// TIA Portal V17 export
// export: Created 2025-08-05T09:36:00.5262225Z, ExportSetting WithDefaults, DisplayName Totally Integrated Automation Portal, DisplayVersion V17, DisplayName TIA Portal Openness, DisplayVersion V17, DisplayName TIA Portal Version Control Interface, DisplayVersion V17, DisplayName SINAMICS Startdrive Advanced, DisplayVersion V17, DisplayName SINAMICS Startdrive G130, G150, S120, S150, SINAMICS MV, S210, DisplayVersion V17, DisplayName SINAMICS Startdrive G110M, G120, G120C, G120D, G120P, G115D, DisplayVersion V17, DisplayName STEP 7 Professional, DisplayVersion V17, DisplayName STEP 7 Safety, DisplayVersion V17, DisplayName WinCC Advanced, DisplayVersion V17
TYPE "typeUserLevel"
TITLE = HMI user levels / HMI Benutzerstufen
// HMI user levels [V 01.00 | Kernel_V2] / HMI Benutzerstufen [V 01.00 | Kernel_V2]
// stored: IsFailsafeCompliant false
   STRUCT
      userLevelBitByBit : Struct   // Aktives Benutzerlevel Bitweise / Active user level bit by bit
         level1 : Bool;   // Benutzerlevel 1 (Admin) / User level 1 (Admin)
         level2 : Bool;   // Benutzerlevel 2 (Hersteller) / User level 2 (Manufacturer)
         level3 : Bool;   // Benutzerlevel 3 (Instandhaltung) / User level 3 (Maintenance)
         level4 : Bool;   // Benutzerlevel 4 (User) / User level 4 (User)
         level5 : Bool;   // Benutzerlevel 5 (Keyswitch 3) / User level 5 (Keyswitch 3)
         level6 : Bool;   // Benutzerlevel 6 (Keyswitch 2) / User level 6 (Keyswitch 2)
         level7 : Bool;   // Benutzerlevel 7 (Keyswicht 1) / User level 7 (Keyswitch 1)
         level8 : Bool;   // Benutzerlevel 8 () / User level 8 ()
      END_STRUCT;
      userLevel : Int;   // Aktives Benutzerlevel / Active user level
      userLevelChanged : Bool;   // Aktives Benutzerlevel gewechselt / Active user level changed
   END_STRUCT;
END_TYPE
